// Mitsubishi GX Works2 project: LRI - PLC - AULA 5   PLC: Q03UDV

PROGRAM MAIN
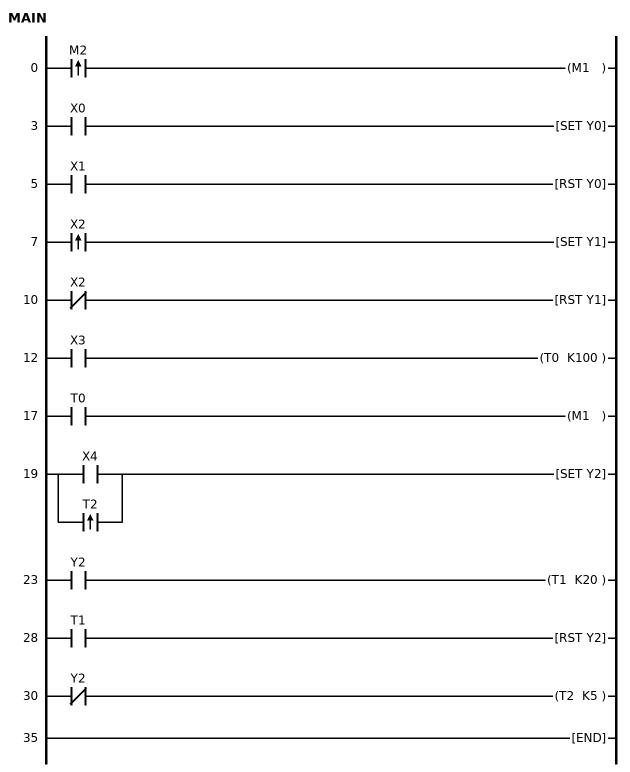
0     LDP     M2
      OUT     M1
3     LD      X0
      SET     Y0
5     LD      X1
      RST     Y0
7     LDP     X2
      SET     Y1
10    LDI     X2
      RST     Y1
12    LD      X3
      OUT     T0 K100
17    LD      T0
      OUT     M1
19    LD      X4
      ORP     T2
      SET     Y2
23    LD      Y2
      OUT     T1 K20
28    LD      T1
      RST     Y2
30    LDI     Y2
      OUT     T2 K5
35    END
END_PROGRAM
